PROGRAM MAIN
VAR
END_VAR

P_CraneControl();

END_PROGRAM

(* stored: Version 1.1.0.1, ProductVersion 3.1.4024.10
   POU MAIN: Id {d407ed84-4ffd-4e3c-9559-a3e35f8925bf}, SpecialFunc None *)
